Staubli VAL3: refresh.pgx

program refresh()
// // page refresh
begin
  if (nKey>=270 and nKey<=278) or use:bUseRefresh==true
    cls()
    call refreshStatic()
    call buildList()
    call refreshDynamic()
    //  nIndex=data:nPage_viewTraj
    if abs(clock()-nRefresh)>nTime
      call refreshDynamic()
    endIf
  endIf
    delay(0)
end
